Fanuc KAREL source: kt00496.KL

PROGRAM KT00496
%STACKSIZE=65535
%PRIORITY=65535
%NOLOCKGROUP
VAR
P1 : XYZWPR
P2 : POSITION
OUT : XYZWPREXT
BEGIN
P1.X=1.0
-- UNRESOLVED_PC line 9 opcodes [49 7E 49 60 7E 4A] marker_code=20
END KT00496
